(* PLC project safeApp1, BrAutomation SafeDESIGNER  5.16.0.0 *)
(* stored: companyURL http://www.br-automation.com, creationDateTime Wed Apr 20 11:11:09 2022 *)

PROGRAM Main
  VAR  (* added by the conversion: wires and edge detectors of the diagram *)
    _AND_S25_OUT : SAFEBOOL;
    _AND_S79_OUT : SAFEBOOL;
    _AND_S35_OUT : SAFEBOOL;
    _AND_S219_OUT : ANY;
    _AND_S233_OUT : ANY;
    _AND_S158_OUT : SAFEBOOL;
  END_VAR

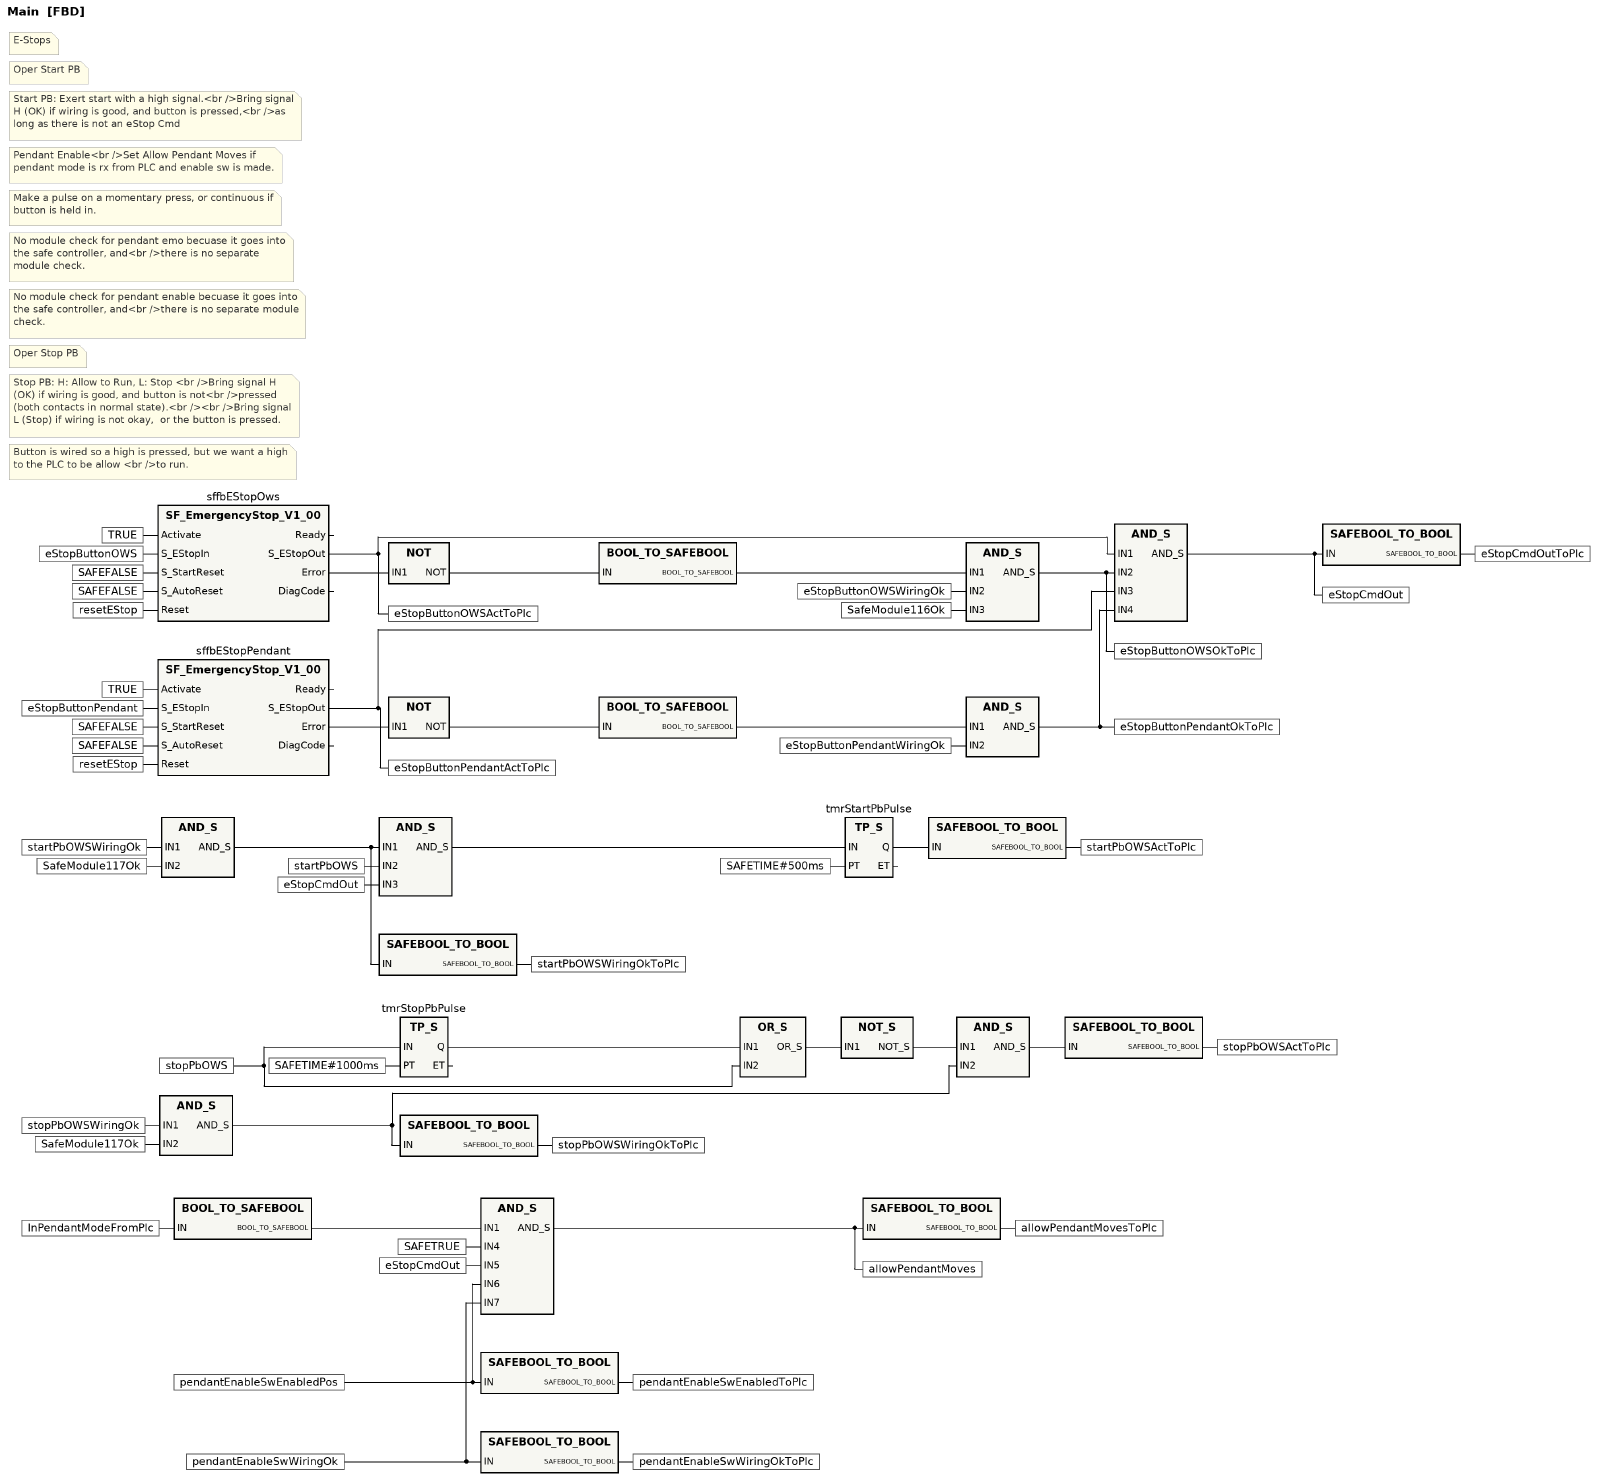
(* FBD diagram, written out as Structured Text *)
(* E-Stops *)
sffbEStopOws(Activate := TRUE, S_EStopIn := eStopButtonOWS, S_StartReset := SAFEFALSE, S_AutoReset := SAFEFALSE, Reset := resetEStop);
eStopButtonOWSActToPlc := sffbEStopOws.S_EStopOut;
_AND_S25_OUT := AND_S(BOOL_TO_SAFEBOOL(NOT sffbEStopOws.Error), eStopButtonOWSWiringOk, SafeModule116Ok);
eStopButtonOWSOkToPlc := _AND_S25_OUT;
sffbEStopPendant(Activate := TRUE, S_EStopIn := eStopButtonPendant, S_StartReset := SAFEFALSE, S_AutoReset := SAFEFALSE, Reset := resetEStop);
_AND_S79_OUT := AND_S(BOOL_TO_SAFEBOOL(NOT sffbEStopPendant.Error), eStopButtonPendantWiringOk);
_AND_S35_OUT := AND_S(sffbEStopOws.S_EStopOut, _AND_S25_OUT, sffbEStopPendant.S_EStopOut, _AND_S79_OUT);
eStopCmdOut := _AND_S35_OUT;
eStopButtonPendantActToPlc := sffbEStopPendant.S_EStopOut;
eStopCmdOutToPlc := SAFEBOOL_TO_BOOL(_AND_S35_OUT);
(* No module check for pendant emo becuase it goes into the safe controller, and<br />there is no separate module check. *)
eStopButtonPendantOkToPlc := _AND_S79_OUT;
(* Oper Start PB *)
(* Start PB: Exert start with a high signal.<br />Bring signal H (OK) if wiring is good, and button is pressed,<br />as long as there is not an eStop Cmd *)
_AND_S219_OUT := AND_S(startPbOWSWiringOk, SafeModule117Ok);
startPbOWSWiringOkToPlc := SAFEBOOL_TO_BOOL(_AND_S219_OUT);
tmrStartPbPulse(IN := AND_S(_AND_S219_OUT, startPbOWS, eStopCmdOut), PT := SAFETIME#500ms);
startPbOWSActToPlc := SAFEBOOL_TO_BOOL(tmrStartPbPulse.Q);
(* Oper Stop PB *)
(* Stop PB: H: Allow to Run, L: Stop <br />Bring signal H (OK) if wiring is good, and button is not<br />pressed (both contacts in normal state).<br /><br />Bring signal L (Stop) if wiring is not okay,  or the button is pressed. *)
(* Make a pulse on a momentary press, or continuous if button is held in. *)
(* Button is wired so a high is pressed, but we want a high to the PLC to be allow <br />to run. *)
tmrStopPbPulse(IN := stopPbOWS, PT := SAFETIME#1000ms);
_AND_S233_OUT := AND_S(stopPbOWSWiringOk, SafeModule117Ok);
stopPbOWSActToPlc := SAFEBOOL_TO_BOOL(AND_S(NOT_S(OR_S(tmrStopPbPulse.Q, stopPbOWS)), _AND_S233_OUT));
stopPbOWSWiringOkToPlc := SAFEBOOL_TO_BOOL(_AND_S233_OUT);
(* Pendant Enable<br />Set Allow Pendant Moves if pendant mode is rx from PLC and enable sw is made. *)
_AND_S158_OUT := AND_S(BOOL_TO_SAFEBOOL(InPendantModeFromPlc), SAFETRUE, eStopCmdOut, pendantEnableSwEnabledPos, pendantEnableSwWiringOk);
allowPendantMoves := _AND_S158_OUT;
allowPendantMovesToPlc := SAFEBOOL_TO_BOOL(_AND_S158_OUT);
(* No module check for pendant enable becuase it goes into the safe controller, and<br />there is no separate module check. *)
pendantEnableSwWiringOkToPlc := SAFEBOOL_TO_BOOL(pendantEnableSwWiringOk);
pendantEnableSwEnabledToPlc := SAFEBOOL_TO_BOOL(pendantEnableSwEnabledPos);
END_PROGRAM
